FUNCTION Greater_Smaller : INT
VAR_INPUT
	nNumber1 : INT;
	nNumber2 : INT;
END_VAR

VAR_OUTPUT
	nGreater : INT;
	nSmaller : INT;
	
END_VAR


IF nNumber1 > nNumber2 THEN
	nGreater := nNumber1;
	nSmaller := nNumber2;

ELSE 
	nGreater := nNumber2;
	nSmaller := nNumber1;	
END_IF

END_FUNCTION

(* stored: Version 1.1.0.1, ProductVersion 3.1.4024.9
   POU Greater_Smaller: Id {39dd69c7-89e8-466a-a7f3-d7600f8ee33c}, SpecialFunc None *)
